TYPE ST_SubsystemErrorStruct :
(**************************************************************************************
 * 	Application		:	BoxControl Framework
 *	Revision		:	$Revision: 404529 $
 *	Revision date	:	$Date: 2018-04-23 08:21:38 +0200 (Mo., 23 Apr 2018) $
 *	Last changed by	:	$Author: b7bolm $
 *	URL				:	$URL: http://almscdc.swisslog.com/repo/SWPD/Development/BoxControlFramework/20_Release/trunk/01_Software/BCF/BCF/JumpStart/20_Product/10_App/15_Subsystem/10_Lib/10_Conv/01_DUTs/ST_SubSystemErrorStruct.TcDUT $
 *
 *	Purpose			:	Group error structure - Contains all information for the
 *						error handling.
 *
 * ------------------------------------------------------------------------------------
 *	Copyright Swisslog [IP AG], Switzerland. All rights reserved.
 * 
 * ------------------------------------------------------------------------------------
 *	
 * 	Revision History: 
 *
 * 	VERSION			DATE			INITIALS			DESCRIPTION
 *	0.1				01.01.2001		swl					Example
 *
 **************************************************************************************)
STRUCT
	ErrorState				: E_ErrorState; // Ongoing module error state
	Error					: ST_ErrorDataSet; // Ongoing reported error
	DataSetIdx				: INT; // Choosen error set index
	ErrorDataSet			: ARRAY [1..NUMBER_OF_ERROR_SETS] OF ST_ErrorDataSet; // Overview about all message sets
	ExternalError			: ST_ErrorDataSet; // External error, Can be set customized or by control code
	GroupErrorPending		: BOOL; // A group is in error state
END_STRUCT
END_TYPE

(* stored: Version 1.1.0.1, ProductVersion 3.1.4022.12
   DUT ST_SubSystemErrorStruct: Id {762585a1-b20c-46aa-86d3-2a7549c061d0} *)
